{attribute 'reflection'} 
FUNCTION_BLOCK FB_DigitalInput IMPLEMENTS I_DigitalChannel
VAR_INPUT
	tDebounce:			TIME:= T#50MS;
END_VAR
VAR_OUTPUT
END_VAR
VAR

	sName:				STRING(25);	// Equipment ID
	Channel			AT%I*: BOOL;	// Link to input
	fbDebounce:		FB_Debounce;
END_VAR

// https://github.com/PeterZerlauth/Tc3_Component
fbDebounce(bInput:= Channel, tTime:= tDebounce);

PROPERTY PUBLIC P_Name : String(25)
GET
P_Name:= sName;
END_GET
END_PROPERTY

PROPERTY P_State : EPlcMappingStatus
GET
P_State:= F_GetMappingStatus(ADR(Channel), SIZEOF(BOOL));
END_GET
END_PROPERTY

PROPERTY PUBLIC P_Value : bool
GET
P_Value:= fbDebounce.bValue;
END_GET
SET // PUBLIC
END_SET
END_PROPERTY

END_FUNCTION_BLOCK

(* stored: Version 1.1.0.1
   POU FB_DigitalInput: Id {8904ca26-c33a-0d5e-01bd-927c832f4cd0}, SpecialFunc None
   Property P_Name: Id {d2592e33-0c09-00ed-2a19-2a2ac1387854}
   Get Get: Id {db03f916-1db4-0ef0-2610-a102e9e38d81}
   Property P_State: Id {c3d8c2a3-d582-03a1-3305-487cd866c231}
   Get Get: Id {d84261ad-8c83-064f-0dc4-445397d3c6cc}
   Property P_Value: Id {eb10c2b4-f572-0e2d-2bec-edb3aca0020c}
   Get Get: Id {0af5f71f-a62f-0bc9-1f1b-442ea0defb72}
   Set Set: Id {a5ae33fe-bcc6-09a5-0371-0da6975e192e} *)
